VISUALIZATION VI_CmdHistorySide  // 2x2
END_VISUALIZATION

(* stored: Version 1.1.0.1, ProductVersion 3.1.4024.9
   Visu VI_CmdHistorySide: Id {8164e9ab-59e2-4e22-8172-cc973f954056} *)
